// TIA Portal V20 export
DATA_BLOCK "DB_OPC_Alarms"   // DB117
{ S7_Optimized_Access := 'TRUE' }
// stored: MemoryReserve 100
   VAR
      NumberOfActiveAlarms : DInt;
      ActiveAlarms : Array[0..50] of "UDT_Alarms";
      Update { S7_SetPoint := 'True'} : Byte;   // A modifier lors d'un Acknowledge
   END_VAR
BEGIN
END_DATA_BLOCK
